TYPE In_16_To_PLC :
STRUCT
	In AT %Q*:ARRAY [1..16] OF BOOL;
END_STRUCT
END_TYPE

(* stored: Version 1.1.0.1, ProductVersion 3.1.4024.14
   DUT In_16_To_PLC: Id {fd97ada8-8eb8-49e0-8229-929af9611b0f} *)
